// TIA Portal V17 export
// export: Created 2024-08-07T21:43:58.2232017Z, ExportSetting WithDefaults, DisplayName Totally Integrated Automation Portal, DisplayVersion V17 Update 7, DisplayName TIA Portal Openness, DisplayVersion V17 Update 7, DisplayName TIA Portal Version Control Interface, DisplayVersion V17, DisplayName SINAMICS Startdrive Advanced, DisplayVersion V17 SP2, DisplayName SINAMICS Startdrive G110M, G120, G120C, G120D, G120P, G115D, DisplayVersion V17 SP2, DisplayName SINAMICS Startdrive G130, G150, S120, S150, SINAMICS MV, S210, DisplayVersion V17 SP2, DisplayName STEP 7 Professional, DisplayVersion V17 Update 7, DisplayName STEP 7 Safety, DisplayVersion V17 Update 6, DisplayName WinCC Advanced / Unified PC, DisplayVersion V17 Update 7
FUNCTION "FC_READING_MAIN" : Void   // FC304, LAD
{ S7_Optimized_Access := 'TRUE' }
VERSION : 0.1
// stored: AutoNumber false, IsIECCheckEnabled false, SetENOAutomatically false, UDAEnableTagReadback false
BEGIN

REGION Network 1: Dataman readers block calls
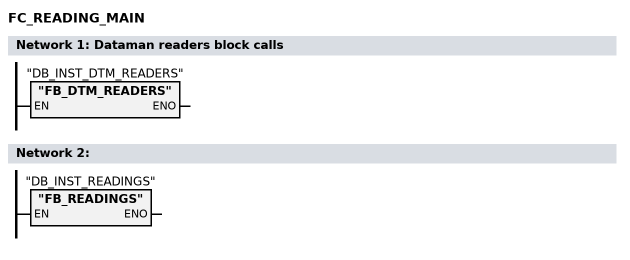
   RUNG wire#powerrail
      "DB_INST_DTM_READERS"()
   END_RUNG
   // the same network as SCL:
   "DB_INST_DTM_READERS"();   // "FB_DTM_READERS"
END_REGION

REGION Network 2
   RUNG wire#powerrail
      "DB_INST_READINGS"()
   END_RUNG
   // the same network as SCL:
   "DB_INST_READINGS"();   // "FB_READINGS"
END_REGION
END_FUNCTION
